ORGANIZATION_BLOCK MAIN:OB1
TITLE=Pulse Test Program
BEGIN
Network 1
LD     SM0.1
MOVW   0, VW100
MOVW   0, VW102

Network 2
LD     I0.0
EU
INCW   VW100

Network 3
LD     I0.1
EU
INCW   VW102

END_ORGANIZATION_BLOCK
